FUNCTION_BLOCK FB_EventLogger
VAR_INPUT
END_VAR
VAR_OUTPUT
END_VAR
VAR
	buffer_counter:INT;
	EventBuffer: ARRAY[1..MAXIMUN_SIZE_OF_EVENT_BUFFR] OF ST_Event;
	EventBuffer_clear: ARRAY[1..MAXIMUN_SIZE_OF_EVENT_BUFFR] OF ST_Event;
	EventBufferIndex:INT:=0;
END_VAR
VAR CONSTANT
	MAXIMUN_SIZE_OF_EVENT_BUFFR:INT :=100;
END_VAR

METHOD IsEventBufferFull : BOOL
VAR_INPUT
END_VAR
IF (EventBufferIndex+1) > MAXIMUN_SIZE_OF_EVENT_BUFFR THEN
	EventBuffer:=EventBuffer_clear;
	EventBufferIndex:=0 ;
	//IsEventBufferFull:=TRUE; 
END_IF
IsEventBufferFull:=FALSE;
END_METHOD

(* returns false if not succesfull*) 
METHOD PUBLIC mAdd : BOOL
VAR_INPUT
	
END_VAR

VAR
	arrDataToWrite: INT;
END_VAR

IF NOT IsEventBufferFull() THEN
	EventBufferIndex:=EventBufferIndex+1;
	EventBuffer[EventBufferIndex].eEventType:=gEventType;
	EventBuffer[EventBufferIndex].eEventSeverity:=gEventSeverity;
	EventBuffer[EventBufferIndex].nEventIdentity:=gEventIdentity;
	EventBuffer[EventBufferIndex].sEventName:=gEventName;
	EventBuffer[EventBufferIndex].sEventText:=gEventText;
	UpdateEventTimestampWithSystemTime (stEvent:=EventBuffer[EventBufferIndex]); 
	sEventTime:= DT_TO_STRING (EventBuffer[EventBufferIndex].dtTimestamp);
	mAdd:=TRUE ;
ELSE
	mAdd:=FALSE;
END_IF
END_METHOD

END_FUNCTION_BLOCK

(* stored: Version 1.1.0.1, ProductVersion 3.1.4024.12
   POU FB_EventLogger: Id {ce2a722b-5878-4631-9052-9e37560196c4}, SpecialFunc None
   Method IsEventBufferFull: Id {8f82d951-cb10-4ede-902a-fe0225981d02}
   Method mAdd: Id {89335789-7a03-417e-9cd7-03d6b2902c98} *)
